FUNCTION_BLOCK OnOffDevice IMPLEMENTS I_DigitalDevice
VAR
	Q AT%Q* : BOOL;
END_VAR

PROPERTY Status : BOOL
GET

	Status	:=	Q;
END_GET
END_PROPERTY

METHOD TurnOff
VAR_INPUT
END_VAR

	Q	:=	FALSE;
END_METHOD

METHOD TurnOn
VAR_INPUT
END_VAR

	Q	:=	TRUE;
END_METHOD

END_FUNCTION_BLOCK

(* stored: Version 1.1.0.1, ProductVersion 3.1.4024.13
   POU OnOffDevice: Id {35b57e29-fc05-43f7-9e56-cc829be85280}, SpecialFunc None
   Property Status: Id {6c52272f-94bf-4a1d-838f-365d773da574}
   Get Get: Id {5030d7d7-00d0-4cb9-b97d-fa41290f95ac}
   Method TurnOff: Id {3a2a1b56-7964-4e35-b443-b51324af685f}
   Method TurnOn: Id {6aab5918-cecd-4e5a-a891-ecb09c028d24} *)
